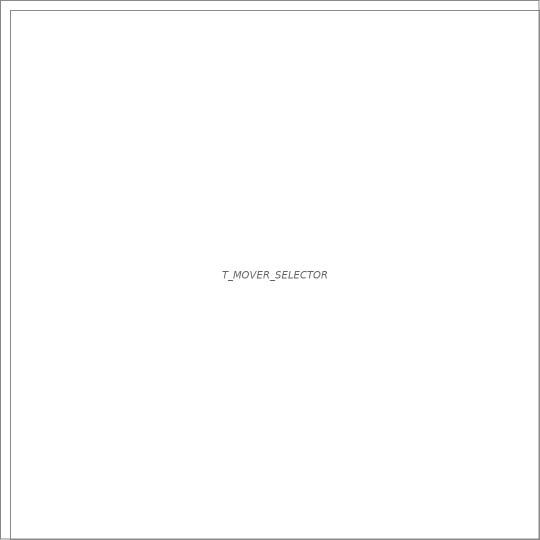
VISUALIZATION SELECTOR_VISU  // 540x540
    Frame (10,10 530x530)
        shows T_MOVER_SELECTOR(Control := GVL_XTS.SelectorCtrl, State := GVL_XTS.SelectorState, sState := MAIN.sSelectorState, sResult := MAIN.sSelectorResult)
END_VISUALIZATION

(* stored: Version 1.1.0.1, ProductVersion 3.1.4026.20
   Visu SELECTOR_VISU: Id {a33d2ec5-ecce-4edd-ae82-53d4a1811924} *)
